(* Logix 5000 project; controller PLC_1_Week_5_Parking_Lot vendor 1 type 14 code 96 rev 30.11; software revision 30.01 *)

TASK MainTask (continuous, watchdog 500 ms) : MainProgram

MODULES
   Local : vendor 1 type 14 code 96 (ICP 2, rev 30.11)
END_MODULES

PROGRAM MainProgram   (* main routine MainRoutine *)
VAR
   CAR_IN_OUT : COUNTER := (PRE := 8);
   CAR_OUT : COUNTER := (PRE := 8);
   CLOSE_ENTRANCE : TIMER := (PRE := 20000);
   CLOSE_EXIT : TIMER := (PRE := 20000);
   ENTRANCE_GATE : BOOL;
   EXIT_GATE : BOOL;
   GREEN_LIGHT : BOOL;
   KEY_CARD : BOOL;   // Key Card
   LOT_FULL : BOOL;
   POWER : BOOL;
   S1 : BOOL;   // Entrance Proximity
   S2 : BOOL;   // In Proximity
   S3 : BOOL;   // Out Proximity
   S4 : BOOL;   // Exit Proximity
   START : BOOL;
   STOP : BOOL;
END_VAR

ROUTINE MainRoutine   (* ladder *)
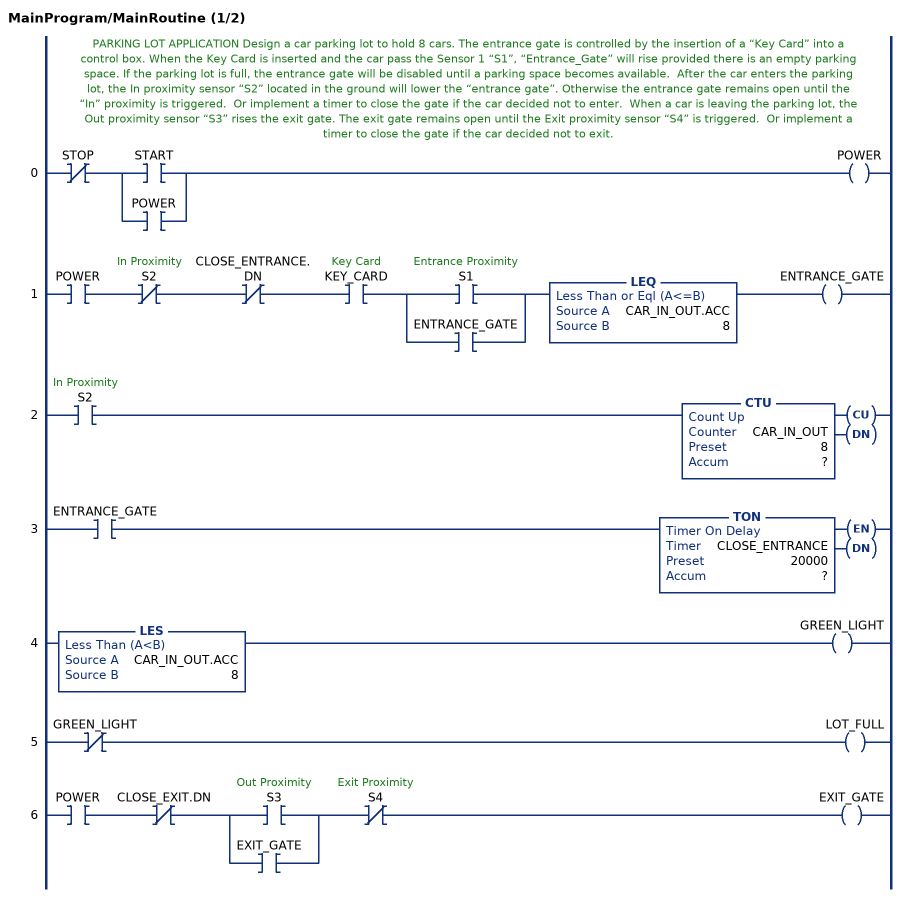
   // PARKING LOT APPLICATION Design a car parking lot to hold 8 cars. The entrance gate is controlled by the insertion of a “Key Card” into a control box. When the Key Card is inserted and the car pass the Sensor 1 “S1”, “Entrance_Gate” will rise provided there is an empty parking space. If the parking lot is full, the entrance gate will be disabled until a parking space becomes available.  After the car enters the parking lot, the In proximity sensor “S2” located in the ground will lower the “entrance gate”. Otherwise the entrance gate remains open until the “In” proximity is triggered.  Or implement a timer to close the gate if the car decided not to enter.  When a car is leaving the parking lot, the Out proximity sensor “S3” rises the exit gate. The exit gate remains open until the Exit proximity sensor “S4” is triggered.  Or implement a timer to close the gate if the car decided not to exit.
   0: XIO(STOP)[XIC(START) ,XIC(POWER) ]OTE(POWER);
   1: XIC(POWER)XIO(S2)XIO(CLOSE_ENTRANCE.DN)XIC(KEY_CARD)[XIC(S1) ,XIC(ENTRANCE_GATE) ]LEQ(CAR_IN_OUT.ACC,8)OTE(ENTRANCE_GATE);
   2: XIC(S2)CTU(CAR_IN_OUT,?,?);
   3: XIC(ENTRANCE_GATE)TON(CLOSE_ENTRANCE,?,?);
   4: LES(CAR_IN_OUT.ACC,8)OTE(GREEN_LIGHT);
   5: XIO(GREEN_LIGHT)OTE(LOT_FULL);
   6: XIC(POWER)XIO(CLOSE_EXIT.DN)[XIC(S3) ,XIC(EXIT_GATE) ]XIO(S4)OTE(EXIT_GATE);
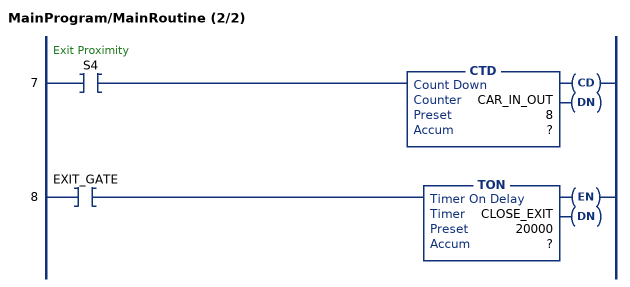
   7: XIC(S4)CTD(CAR_IN_OUT,?,?);
   8: XIC(EXIT_GATE)TON(CLOSE_EXIT,?,?);
END_ROUTINE
END_PROGRAM
